Universal Robots URScript: 00C_04_Qu_BoXian.script

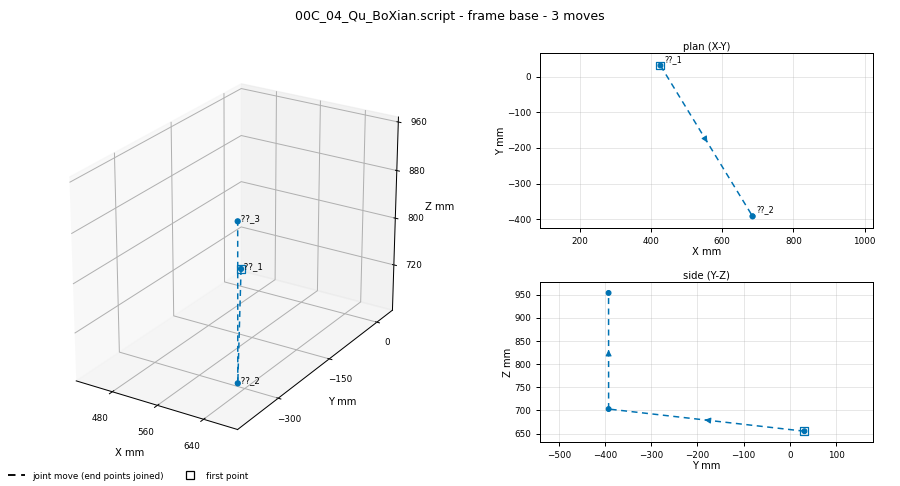
[picture p0: tool path of 00C_04_Qu_BoXian.script in frame base, 3 of 3 moves have a stored position in this frame; points joined in program order, loops and branches not executed]
def P00C_04_Qu_BoXian():
  set_standard_analog_input_domain(0, 1)
  set_standard_analog_input_domain(1, 1)
  set_tool_analog_input_domain(0, 1)
  set_tool_analog_input_domain(1, 1)
  set_analog_outputdomain(0, 0)
  set_analog_outputdomain(1, 0)
  set_tool_voltage(0)
  set_input_actions_to_default()
  set_tcp(p[-0.06448999999999999,0.0207,0.28314999999999996,0.0,0.0,1.5902])
  set_payload(8.0)
  set_safety_mode_transition_hardness(1)
  set_gravity([0.0, 0.0, 9.82])
  $ 1 "机器人程序"
  $ 2 "MoveJ"
  $ 3 "路点_1"
  set_tcp(p[-8.5E-4,0.01448,0.31003,0.0,0.0,-0.3645])
  movej(get_inverse_kin(p[.426729406315, .031412478142, .655040505919, -.007982663310, .061422349307, -1.298956988393], qnear=[0.5012885332107544, -1.4665511290179651, -2.670982901250021, -0.6037114302264612, -1.524388615285055, -3.0076070467578333]), a=0.6981317007977318, v=0.5235987755982988)
  $ 4 "路点_2"
  set_tcp(p[-8.5E-4,0.01448,0.31003,0.0,0.0,-0.3645])
  movej(get_inverse_kin(p[.685521945712, -.392102168779, .702949784238, -.014120828226, .061722199037, -1.493857918143], qnear=[-0.3257835547076624, -1.9238598982440394, -1.9763367811786097, -0.8674381414996546, -1.5680936018573206, -2.3762980143176478]), a=0.6981317007977318, v=0.5235987755982988)
  $ 5 "路点_3"
  set_tcp(p[-8.5E-4,0.01448,0.31003,0.0,0.0,-0.3645])
  movej(get_inverse_kin(p[.685528203690, -.392195154123, .954076360947, -.014202838530, .061808046631, -1.493936076535], qnear=[-0.32687551179994756, -1.7050188223468226, -1.7463038603412073, -1.3163984457599085, -1.5682733694659632, -2.3786962668048304]), a=0.6981317007977318, v=0.5235987755982988)
end
